// TIA Portal V20 export
TYPE "LER_typeMobileRFIDConfiguration"
// stored: Access Published
   STRUCT
      referenceDesignator : WString[25];
      connectData : TCON_IP_v4;
   END_STRUCT;
END_TYPE
